
(* ===== HMI "HMI_RT_4" =====

HMI tags "PAC2200"
   "Frequency" : Real, internal   // Frequency [Hz]
   "I_Avg" : Real, internal   // Average current [A]
   "I_N" : Real, internal   // Neutral current [A]
   "I1" : Real, internal   // Current L1 [A]
   "I2" : Real, internal   // Current L2 [A]
   "I3" : Real, internal   // Current L3 [A]
   "P_Total_Exp" : Real, internal   // Active energy export [Wh]
   "P_Total_Imp" : Real, internal   // Active energy import [Wh]
   "Q_Total_Exp" : Real, internal   // Reactive energy export [varh]
   "Q_Total_Imp" : Real, internal   // Reactive energy import [varh]
   "P_L1" : Real, internal   // Active power L1 [W]
   "P_L2" : Real, internal   // Active power L2 [W]
   "P_L3" : Real, internal   // Active power L3 [W]
   "P_Total" : Real, internal   // Total active power [W]
   "Q_L1" : Real, internal   // Reactive power L1 [var]
   "Q_L2" : Real, internal   // Reactive power L2 [var]
   "Q_L3" : Real, internal   // Reactive power L3 [var]
   "Q_Total" : Real, internal   // Total reactive power [var]
   "S_L1" : Real, internal   // Apparent power L1 [VA]
   "S_L2" : Real, internal   // Apparent power L2 [VA]
   "S_L3" : Real, internal   // Apparent power L3 [VA]
   "S_Total" : Real, internal   // Total apparent power [VA]
   "PF_L1" : Real, internal   // Power factor L1 []
   "PF_L2" : Real, internal   // Power factor L2 []
   "PF_L3" : Real, internal   // Power factor L3 []
   "PF_Tot" : Real, internal   // Total power factor []
   "L1_L2" : Real, internal   // Voltage L1-L2 [V]
   "L1_N" : Real, internal   // Voltage L1-N [V]
   "L2_L3" : Real, internal   // Voltage L2-L3 [V]
   "L2_N" : Real, internal   // Voltage L2-N [V]
   "L3_L1" : Real, internal   // Voltage L3-L1 [V]
   "L3_N" : Real, internal   // Voltage L3-N [V]
   "LL_Avg" : Real, internal   // Average voltage L-L [V]
   "LN_Avg" : Real, internal   // Average voltage L-N [V]
   "Connection_State" : Int, internal   // Modbus TCP/IP connection state 0: OFFLINE; 1: ONLINE;
   "Enable" : Bool, internal   // Modbus TCP/IP request enable
   "IPv4" : WString[254], internal   // IPv4 address
   "Polling_Timestamp" : WString[254], internal   // Last received data
   "Port_Number" : Int, internal   // Modbus TCP/IP port number
   "Unit_Id" : Int, internal   // Modbus TCP/IP unit ID
   "Device_Type" : Int, internal   // Sentron device type
   "Error" : Int, internal   // Modbus TCP/IP error 0: ACK; 1: NACK
   "Error_Code" : Int, internal   // Modbus TCP/IP error code
   "Error_Code_Desc" : WString[254], internal   // Modbus TCP/IP error code description
*)